% RSLogix 500 project PROJECT6.RSS, saved by version 8.30.00.16 %
PROJECT "PROJECT6"    % processor: Bul.1763 MicroLogix 1100 Series B %

PROGRAM FILES
  LAD 2 "MAIN"  4 rungs
  LAD 3 "DI/DO"  3 rungs
  LAD 4 "CONTROL"  10 rungs

DATA FILES
  O0 OUTPUT  5 elements
  I1 INPUT  7 elements
  S2 STATUS  66 elements
  B3 BINARY  1 elements
  T4 TIMER  1 elements
  C5 COUNTER  3 elements
  R6 CONTROL  1 elements
  N7 INTEGER  4 elements
  F8 FLOAT  1 elements

LADDER 2 "MAIN"
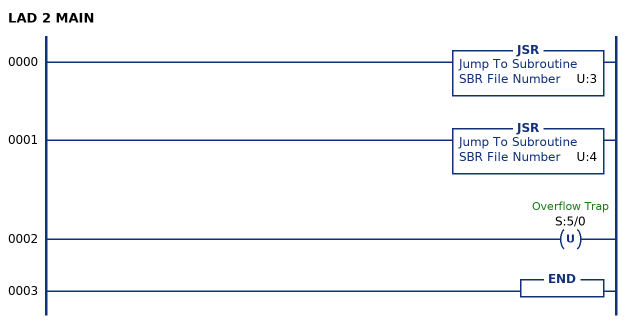
% Rung: 0 %
SOR JSR U:3 EOR
% Rung: 1 %
SOR JSR U:4 EOR
% Rung: 2 %
SOR OTU S:5/0 EOR
%   S:5/0  "Overflow Trap" %
% Rung: 3 %
SOR END EOR

LADDER 3 "DI/DO"
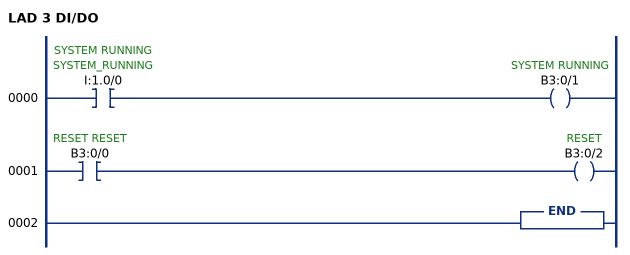
% Rung: 0 %
SOR XIC I:1.0/0 OTE B3:0/1 EOR
%   I:1.0/0  SYSTEM_RUNNING  "SYSTEM RUNNING" %
%   B3:0/1  "SYSTEM RUNNING" %
% Rung: 1 %
SOR XIC B3:0/0 OTE B3:0/2 EOR
%   B3:0/0  RESET  "RESET" %
%   B3:0/2  "RESET" %
% Rung: 2 %
SOR END EOR

LADDER 4 "CONTROL"
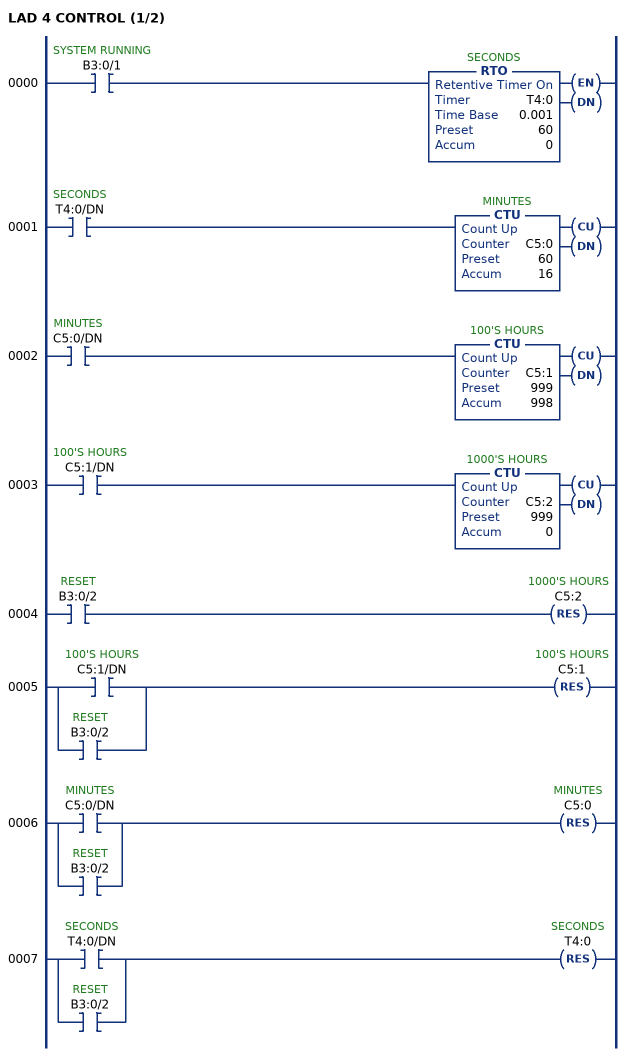
% Rung: 0 %
SOR XIC B3:0/1 RTO T4:0 0.001 60 0 EOR
%   B3:0/1  "SYSTEM RUNNING" %
%   T4:0  "SECONDS" %
% Rung: 1 %
SOR XIC T4:0/DN CTU C5:0 60 16 EOR
%   T4:0  "SECONDS" %
%   C5:0  "MINUTES" %
% Rung: 2 %
SOR XIC C5:0/DN CTU C5:1 999 998 EOR
%   C5:0  "MINUTES" %
%   C5:1  "100'S HOURS" %
% Rung: 3 %
SOR XIC C5:1/DN CTU C5:2 999 0 EOR
%   C5:1  "100'S HOURS" %
%   C5:2  "1000'S HOURS" %
% Rung: 4 %
SOR XIC B3:0/2 RES C5:2 EOR
%   B3:0/2  "RESET" %
%   C5:2  "1000'S HOURS" %
% Rung: 5 %
SOR BST XIC C5:1/DN NXB XIC B3:0/2 BND RES C5:1 EOR
%   C5:1  "100'S HOURS" %
%   B3:0/2  "RESET" %
% Rung: 6 %
SOR BST XIC C5:0/DN NXB XIC B3:0/2 BND RES C5:0 EOR
%   C5:0  "MINUTES" %
%   B3:0/2  "RESET" %
% Rung: 7 %
SOR BST XIC T4:0/DN NXB XIC B3:0/2 BND RES T4:0 EOR
%   T4:0  "SECONDS" %
%   B3:0/2  "RESET" %

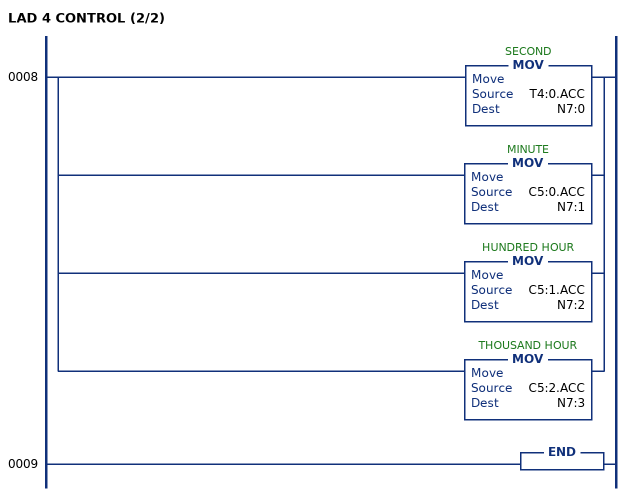
% Rung: 8 %
SOR BST MOV T4:0.ACC N7:0 NXB MOV C5:0.ACC N7:1 NXB MOV C5:1.ACC N7:2 NXB MOV C5:2.ACC N7:3 BND EOR
%   T4:0  "SECONDS" %
%   N7:0  "SECOND" %
%   C5:0.ACC  "MINUTES" %
%   N7:1  "MINUTE" %
%   C5:1  "100'S HOURS" %
%   N7:2  "HUNDRED HOUR" %
%   C5:2  "1000'S HOURS" %
%   N7:3  "THOUSAND HOUR" %
% Rung: 9 %
SOR END EOR

DATA TABLE (non-zero values as saved)
DATA B3
% B3:0 % 0X0002
DATA T4
% .PRE .ACC %
% T4:0 % 60 0
DATA C5
% .PRE .ACC %
% C5:0 % 60 16
% C5:1 % 999 998
% C5:2 % 999 0
